// SIMATIC S7-200 project (STEP 7-Micro/WIN), CPU 222 REL 02.01

SYMBOL_TABLE USER1
CW               I0.0     // ROTAZIONE MOTORE SENSO ORARIO
CCW              I0.1     // ROTAZIONE MOTORE SENSO ANTIORARIO
STOP_            I0.2     // PULSANTE DI ARRESTO
EMERGENZA        I0.3     // EMERGENZA SPENTO
AUX_Q1           I0.4     // PROTEZIONE Q1 INSERITA INTERBLOCCO
AUX_Q2           I0.5     // PROTEZIONE Q2 INSERITA INTERBLOCCO
AUX_Q3           I0.6     // PROTEZIONE Q3 INSERITA INTERBLOCCO
AUX_Q4           I0.7     // PROTEZIONE Q4 INSERITA INTERBLOCCO
AUX_F1           I1.0     // AZIONAMENTO SICUREZZA F1
F4               I1.1     // AZIONAMENTO SICUREZZA RIPRISTINO TERMICA
LEFT             I1.2     // FINECORSA SINISTRA
RIGTH            I1.3     // FINECORSA DESTRA
START_UP         M0.0     // FASE DI AVVIAMENTO
SEL_ORARIO       M0.1     // SELEZIONE SENSO ANTIORARIO
SEL_ANTIORIO     M0.2     // SELEZIONE SENSO ANTIORARIO
FC_RIGHT         M0.3     // FINECORSA DESTRO
FC_LEFT          M0.4     // FINECORSA SINISTRO
ERR_ST_Q3_Q4     M0.5     // INCONGRUO STATO CONTATTORI STELLA TRIANGOLO
ERR_ST_Q1_Q2     M0.6     // INCONGRUO STATO INTERRUTORI LINEA
OK_MARCIA        M0.7     // CONSENSO ALLA MARCIA
CW_CCW           M1.0     // CONTEMPORANEITA CW CCW
Q1               Q0.0     // ROTAZIONE SENSO ORARIO
Q2               Q0.1     // ROTAZIONE SENSO ORARIO
Q3               Q0.2     // COLLEGAMENTO A STELLA
Q4               Q0.3     // COLLEGAMENTO A TRIANGOLO
EL_LEFT          Q0.4     // LAMPADA SEGNALAZIONE LEFT
EL_RIGHT         Q0.5     // LAMPADA SEGALAZIONE RIGHT
END_SYMBOL_TABLE

ORGANIZATION_BLOCK MAIN:OB1
TITLE=SISTEMA MODULARE PER LA SIMULAZIONE DI PROCESSI INDUSTRIALI
// 
// ********** MOTORE TRIFASE***********
// 
BEGIN
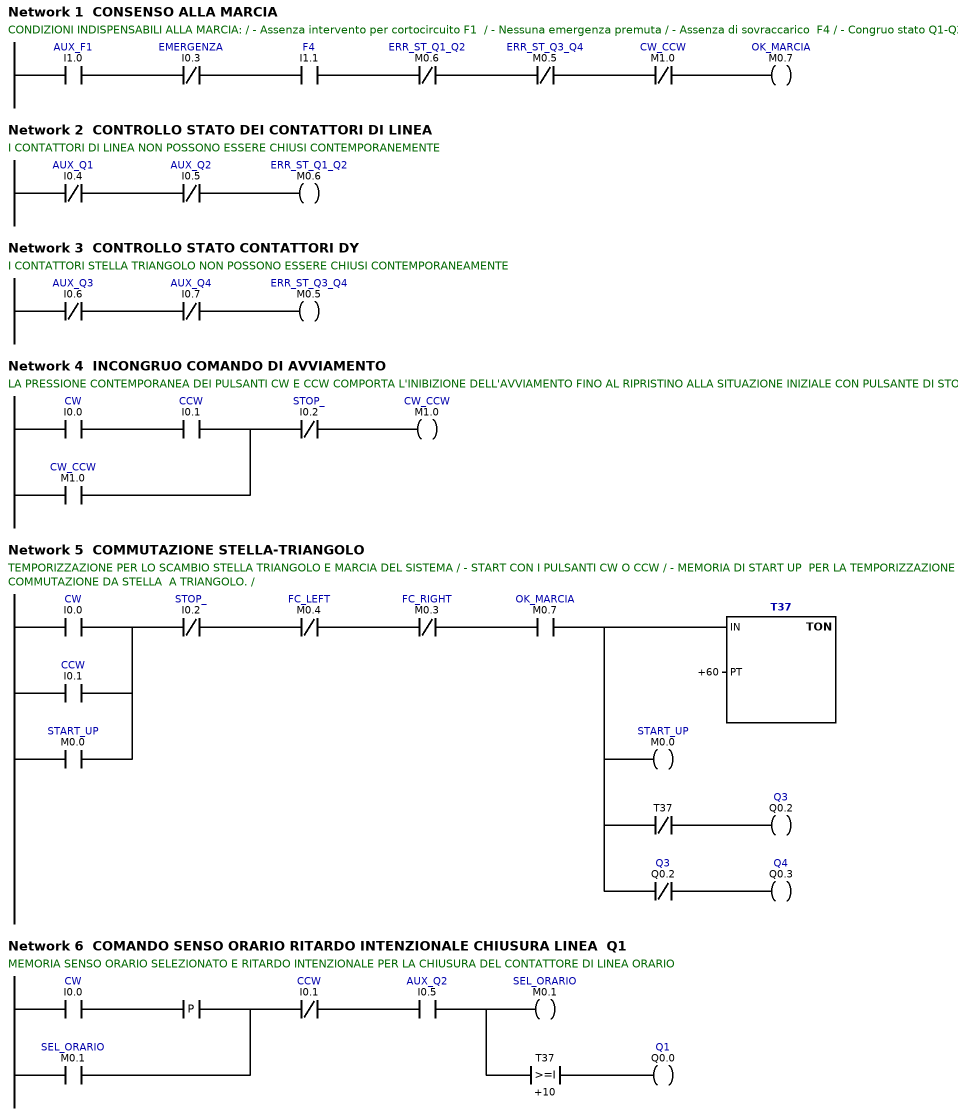
Network 1 // CONSENSO ALLA MARCIA
// CONDIZIONI INDISPENSABILI ALLA MARCIA:
// - Assenza intervento per cortocircuito F1 
// - Nessuna emergenza premuta
// - Assenza di sovraccarico  F4
// - Congruo stato Q1-Q2
// - Congruo stato Q2-Q4
// 
LD     AUX_F1:I1.0
AN     EMERGENZA:I0.3
A      F4:I1.1
AN     ERR_ST_Q1_Q2:M0.6
AN     ERR_ST_Q3_Q4:M0.5
AN     CW_CCW:M1.0
=      OK_MARCIA:M0.7
Network 2 // CONTROLLO STATO DEI CONTATTORI DI LINEA
// I CONTATTORI DI LINEA NON POSSONO ESSERE CHIUSI CONTEMPORANEMENTE
LDN    AUX_Q1:I0.4
AN     AUX_Q2:I0.5
=      ERR_ST_Q1_Q2:M0.6
Network 3 // CONTROLLO STATO CONTATTORI DY
// I CONTATTORI STELLA TRIANGOLO NON POSSONO ESSERE CHIUSI CONTEMPORANEAMENTE
LDN    AUX_Q3:I0.6
AN     AUX_Q4:I0.7
=      ERR_ST_Q3_Q4:M0.5
Network 4 // INCONGRUO COMANDO DI AVVIAMENTO
// LA PRESSIONE CONTEMPORANEA DEI PULSANTI CW E CCW COMPORTA L'INIBIZIONE DELL'AVVIAMENTO FINO AL RIPRISTINO ALLA SITUAZIONE INIZIALE CON PULSANTE DI STOP
LD     CW:I0.0
A      CCW:I0.1
O      CW_CCW:M1.0
AN     STOP_:I0.2
=      CW_CCW:M1.0
Network 5 // COMMUTAZIONE STELLA-TRIANGOLO
// TEMPORIZZAZIONE PER LO SCAMBIO STELLA TRIANGOLO E MARCIA DEL SISTEMA
// - START CON I PULSANTI CW O CCW
// - MEMORIA DI START UP  PER LA TEMPORIZZAZIONE DELL'AVVIAMENTO
// - COMMUTAZIONE DA STELLA  A TRIANGOLO.
// 
LD     CW:I0.0
O      CCW:I0.1
O      START_UP:M0.0
AN     STOP_:I0.2
AN     FC_LEFT:M0.4
AN     FC_RIGHT:M0.3
A      OK_MARCIA:M0.7
LPS
TON    T37, +60
=      START_UP:M0.0
AN     T37
=      Q3:Q0.2
LPP
AN     Q3:Q0.2
=      Q4:Q0.3
Network 6 // COMANDO SENSO ORARIO RITARDO INTENZIONALE CHIUSURA LINEA  Q1
// MEMORIA SENSO ORARIO SELEZIONATO E RITARDO INTENZIONALE PER LA CHIUSURA DEL CONTATTORE DI LINEA ORARIO
LD     CW:I0.0
EU
O      SEL_ORARIO:M0.1
AN     CCW:I0.1
A      AUX_Q2:I0.5
=      SEL_ORARIO:M0.1
AW>=   T37, +10
=      Q1:Q0.0
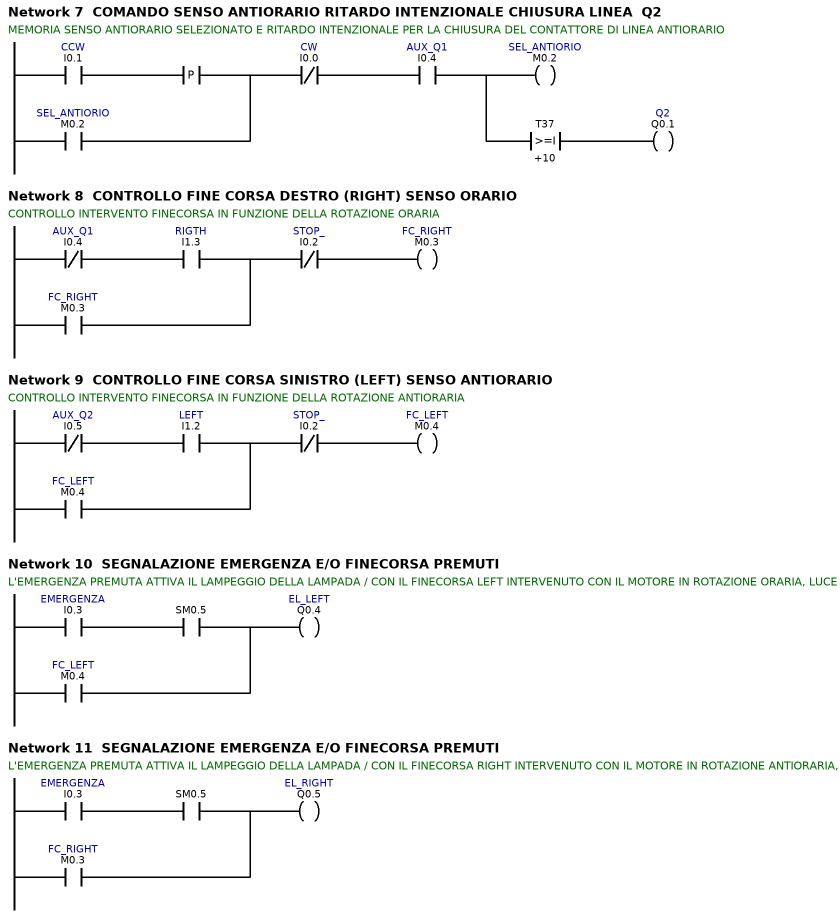
Network 7 // COMANDO SENSO ANTIORARIO RITARDO INTENZIONALE CHIUSURA LINEA  Q2
// MEMORIA SENSO ANTIORARIO SELEZIONATO E RITARDO INTENZIONALE PER LA CHIUSURA DEL CONTATTORE DI LINEA ANTIORARIO
LD     CCW:I0.1
EU
O      SEL_ANTIORIO:M0.2
AN     CW:I0.0
A      AUX_Q1:I0.4
=      SEL_ANTIORIO:M0.2
AW>=   T37, +10
=      Q2:Q0.1
Network 8 // CONTROLLO FINE CORSA DESTRO (RIGHT) SENSO ORARIO
// CONTROLLO INTERVENTO FINECORSA IN FUNZIONE DELLA ROTAZIONE ORARIA
LDN    AUX_Q1:I0.4
A      RIGTH:I1.3
O      FC_RIGHT:M0.3
AN     STOP_:I0.2
=      FC_RIGHT:M0.3
Network 9 // CONTROLLO FINE CORSA SINISTRO (LEFT) SENSO ANTIORARIO
// CONTROLLO INTERVENTO FINECORSA IN FUNZIONE DELLA ROTAZIONE ANTIORARIA
LDN    AUX_Q2:I0.5
A      LEFT:I1.2
O      FC_LEFT:M0.4
AN     STOP_:I0.2
=      FC_LEFT:M0.4
Network 10 // SEGNALAZIONE EMERGENZA E/O FINECORSA PREMUTI
// L'EMERGENZA PREMUTA ATTIVA IL LAMPEGGIO DELLA LAMPADA
// CON IL FINECORSA LEFT INTERVENUTO CON IL MOTORE IN ROTAZIONE ORARIA, LUCE FISSA
LD     EMERGENZA:I0.3
A      SM0.5
O      FC_LEFT:M0.4
=      EL_LEFT:Q0.4
Network 11 // SEGNALAZIONE EMERGENZA E/O FINECORSA PREMUTI
// L'EMERGENZA PREMUTA ATTIVA IL LAMPEGGIO DELLA LAMPADA
// CON IL FINECORSA RIGHT INTERVENUTO CON IL MOTORE IN ROTAZIONE ANTIORARIA, LUCE FISSA
LD     EMERGENZA:I0.3
A      SM0.5
O      FC_RIGHT:M0.3
=      EL_RIGHT:Q0.5
END_ORGANIZATION_BLOCK
